{attribute 'qualified_only'}
VAR_GLOBAL
	BreadIDpicked:INT;
	test:BOOL := FALSE;
END_VAR

(* stored: Version 1.1.0.1, ProductVersion 3.1.4024.15
   GVL HMI: Id {da928412-ba1b-4d91-81c5-38f745b5cd1a} *)
